// TIA Portal V18 export
// export: Created 2026-01-09T11:32:02.097113Z, ExportSetting WithDefaults, DisplayName Totally Integrated Automation Portal, DisplayVersion V18 Update 5, DisplayName TIA Portal Openness, DisplayVersion V18 Update 5, DisplayName TIA Portal Teamcenter Gateway, DisplayVersion V18, DisplayName TIA Portal Version Control Interface, DisplayVersion V18, DisplayName SINAMICS Startdrive Advanced, DisplayVersion V18 SP2 Update 1, DisplayName SINAMICS Startdrive G110M, G120, G120C, G120D, G120P, G115D, DisplayVersion V18 SP2 Update 1, DisplayName SINAMICS Startdrive G130, G150, S120, S150, SINAMICS MV, S210, G220, S200, DisplayVersion V18 SP2 Update 1, DisplayName STEP 7 Professional, DisplayVersion V18 Update 5, DisplayName STEP 7 Safety, DisplayVersion V18, DisplayName WinCC Professional, DisplayVersion V18 Update 5
TagTable "D"
  DnstDataBlock_DP_Status{0} : Bool  (%DB[SysDDBNum].DBX2.0, CPU S71500-2PN_TP700, 1 s)
  DnstDataBlock_DP_Status{1} : Bool  (%DB[SysDDBNum].DBX2.1, CPU S71500-2PN_TP700, 1 s)
  DnstDataBlock_DP_Status{2} : Bool  (%DB[SysDDBNum].DBX2.2, CPU S71500-2PN_TP700, 1 s)
  DnstDataBlock_DP_Status{3} : Bool  (%DB[SysDDBNum].DBX2.3, CPU S71500-2PN_TP700, 1 s)
  DnstDataBlock_DP_Status{4} : Bool  (%DB[SysDDBNum].DBX2.4, CPU S71500-2PN_TP700, 1 s)
  DnstDataBlock_DP_Status{5} : Bool  (%DB[SysDDBNum].DBX2.5, CPU S71500-2PN_TP700, 1 s)
  DnstDataBlock_DP_Status{6} : Bool  (%DB[SysDDBNum].DBX2.6, CPU S71500-2PN_TP700, 1 s)
  DnstDataBlock_DP_Status{7} : Bool  (%DB[SysDDBNum].DBX2.7, CPU S71500-2PN_TP700, 1 s)
  DnstDataBlock_DP_Status{8} : Bool  (%DB[SysDDBNum].DBX3.0, CPU S71500-2PN_TP700, 1 s)
  DnstDataBlock_DP_Status{9} : Bool  (%DB[SysDDBNum].DBX3.1, CPU S71500-2PN_TP700, 1 s)
  DnstDataBlock_DP_Status{10} : Bool  (%DB[SysDDBNum].DBX3.2, CPU S71500-2PN_TP700, 1 s)
  DnstDataBlock_DP_Status{11} : Bool  (%DB[SysDDBNum].DBX3.3, CPU S71500-2PN_TP700, 1 s)
  DnstDataBlock_DP_Status{12} : Bool  (%DB[SysDDBNum].DBX3.4, CPU S71500-2PN_TP700, 1 s)
  DnstDataBlock_DP_Status{13} : Bool  (%DB[SysDDBNum].DBX3.5, CPU S71500-2PN_TP700, 1 s)
  DnstDataBlock_DP_Status{14} : Bool  (%DB[SysDDBNum].DBX3.6, CPU S71500-2PN_TP700, 1 s)
  DnstDataBlock_DP_Status{15} : Bool  (%DB[SysDDBNum].DBX3.7, CPU S71500-2PN_TP700, 1 s)
  DnstDataBlock_DP_Status{16} : Bool  (%DB[SysDDBNum].DBX4.0, CPU S71500-2PN_TP700, 1 s)
  DnstDataBlock_DP_Status{17} : Bool  (%DB[SysDDBNum].DBX4.1, CPU S71500-2PN_TP700, 1 s)
  DnstDataBlock_DP_Status{18} : Bool  (%DB[SysDDBNum].DBX4.2, CPU S71500-2PN_TP700, 1 s)
  DnstDataBlock_DP_Status{19} : Bool  (%DB[SysDDBNum].DBX4.3, CPU S71500-2PN_TP700, 1 s)
  DnstDataBlock_DP_Status{20} : Bool  (%DB[SysDDBNum].DBX4.4, CPU S71500-2PN_TP700, 1 s)
  DnstDataBlock_DP_Status{21} : Bool  (%DB[SysDDBNum].DBX4.5, CPU S71500-2PN_TP700, 1 s)
  DnstDataBlock_DP_Status{22} : Bool  (%DB[SysDDBNum].DBX4.6, CPU S71500-2PN_TP700, 1 s)
  DnstDataBlock_DP_Status{23} : Bool  (%DB[SysDDBNum].DBX4.7, CPU S71500-2PN_TP700, 1 s)
  DnstDataBlock_DP_Status{24} : Bool  (%DB[SysDDBNum].DBX5.0, CPU S71500-2PN_TP700, 1 s)
  DnstDataBlock_DP_Status{25} : Bool  (%DB[SysDDBNum].DBX5.1, CPU S71500-2PN_TP700, 1 s)
  DnstDataBlock_DP_Status{26} : Bool  (%DB[SysDDBNum].DBX5.2, CPU S71500-2PN_TP700, 1 s)
  DnstDataBlock_DP_Status{27} : Bool  (%DB[SysDDBNum].DBX5.3, CPU S71500-2PN_TP700, 1 s)
  DnstDataBlock_DP_Status{28} : Bool  (%DB[SysDDBNum].DBX5.4, CPU S71500-2PN_TP700, 1 s)
  DnstDataBlock_DP_Status{29} : Bool  (%DB[SysDDBNum].DBX5.5, CPU S71500-2PN_TP700, 1 s)
  DnstDataBlock_DP_Status{30} : Bool  (%DB[SysDDBNum].DBX5.6, CPU S71500-2PN_TP700, 1 s)
  DnstDataBlock_DP_Status{31} : Bool  (%DB[SysDDBNum].DBX5.7, CPU S71500-2PN_TP700, 1 s)
  DnstDataBlock_DP_Status{32} : Bool  (%DB[SysDDBNum].DBX6.0, CPU S71500-2PN_TP700, 1 s)
  DnstDataBlock_DP_Status{33} : Bool  (%DB[SysDDBNum].DBX6.1, CPU S71500-2PN_TP700, 1 s)
  DnstDataBlock_DP_Status{34} : Bool  (%DB[SysDDBNum].DBX6.2, CPU S71500-2PN_TP700, 1 s)
  DnstDataBlock_DP_Status{35} : Bool  (%DB[SysDDBNum].DBX6.3, CPU S71500-2PN_TP700, 1 s)
  DnstDataBlock_DP_Status{36} : Bool  (%DB[SysDDBNum].DBX6.4, CPU S71500-2PN_TP700, 1 s)
  DnstDataBlock_DP_Status{37} : Bool  (%DB[SysDDBNum].DBX6.5, CPU S71500-2PN_TP700, 1 s)
  DnstDataBlock_DP_Status{38} : Bool  (%DB[SysDDBNum].DBX6.6, CPU S71500-2PN_TP700, 1 s)
  DnstDataBlock_DP_Status{39} : Bool  (%DB[SysDDBNum].DBX6.7, CPU S71500-2PN_TP700, 1 s)
  DnstDataBlock_DP_Status{40} : Bool  (%DB[SysDDBNum].DBX7.0, CPU S71500-2PN_TP700, 1 s)
  DnstDataBlock_DP_Status{41} : Bool  (%DB[SysDDBNum].DBX7.1, CPU S71500-2PN_TP700, 1 s)
  DnstDataBlock_DP_Status{42} : Bool  (%DB[SysDDBNum].DBX7.2, CPU S71500-2PN_TP700, 1 s)
  DnstDataBlock_DP_Status{43} : Bool  (%DB[SysDDBNum].DBX7.3, CPU S71500-2PN_TP700, 1 s)
  DnstDataBlock_DP_Status{44} : Bool  (%DB[SysDDBNum].DBX7.4, CPU S71500-2PN_TP700, 1 s)
  DnstDataBlock_DP_Status{45} : Bool  (%DB[SysDDBNum].DBX7.5, CPU S71500-2PN_TP700, 1 s)
  DnstDataBlock_DP_Status{46} : Bool  (%DB[SysDDBNum].DBX7.6, CPU S71500-2PN_TP700, 1 s)
  DnstDataBlock_DP_Status{47} : Bool  (%DB[SysDDBNum].DBX7.7, CPU S71500-2PN_TP700, 1 s)
  DnstDataBlock_DP_Status{48} : Bool  (%DB[SysDDBNum].DBX8.0, CPU S71500-2PN_TP700, 1 s)
  DnstDataBlock_DP_Status{49} : Bool  (%DB[SysDDBNum].DBX8.1, CPU S71500-2PN_TP700, 1 s)
  DnstDataBlock_DP_Status{50} : Bool  (%DB[SysDDBNum].DBX8.2, CPU S71500-2PN_TP700, 1 s)
  DnstDataBlock_DP_Status{51} : Bool  (%DB[SysDDBNum].DBX8.3, CPU S71500-2PN_TP700, 1 s)
  DnstDataBlock_DP_Status{52} : Bool  (%DB[SysDDBNum].DBX8.4, CPU S71500-2PN_TP700, 1 s)
  DnstDataBlock_DP_Status{53} : Bool  (%DB[SysDDBNum].DBX8.5, CPU S71500-2PN_TP700, 1 s)
  DnstDataBlock_DP_Status{54} : Bool  (%DB[SysDDBNum].DBX8.6, CPU S71500-2PN_TP700, 1 s)
  DnstDataBlock_DP_Status{55} : Bool  (%DB[SysDDBNum].DBX8.7, CPU S71500-2PN_TP700, 1 s)
  DnstDataBlock_DP_Status{56} : Bool  (%DB[SysDDBNum].DBX9.0, CPU S71500-2PN_TP700, 1 s)
  DnstDataBlock_DP_Status{57} : Bool  (%DB[SysDDBNum].DBX9.1, CPU S71500-2PN_TP700, 1 s)
  DnstDataBlock_DP_Status{58} : Bool  (%DB[SysDDBNum].DBX9.2, CPU S71500-2PN_TP700, 1 s)
  DnstDataBlock_DP_Status{59} : Bool  (%DB[SysDDBNum].DBX9.3, CPU S71500-2PN_TP700, 1 s)
  DnstDataBlock_DP_Status{60} : Bool  (%DB[SysDDBNum].DBX9.4, CPU S71500-2PN_TP700, 1 s)
  DnstDataBlock_DP_Status{61} : Bool  (%DB[SysDDBNum].DBX9.5, CPU S71500-2PN_TP700, 1 s)
  DnstDataBlock_DP_Status{62} : Bool  (%DB[SysDDBNum].DBX9.6, CPU S71500-2PN_TP700, 1 s)
  DnstDataBlock_DP_Status{63} : Bool  (%DB[SysDDBNum].DBX9.7, CPU S71500-2PN_TP700, 1 s)
  DnstDataBlock_DP_Status{64} : Bool  (%DB[SysDDBNum].DBX10.0, CPU S71500-2PN_TP700, 1 s)
  DnstDataBlock_DP_Status{65} : Bool  (%DB[SysDDBNum].DBX10.1, CPU S71500-2PN_TP700, 1 s)
  DnstDataBlock_DP_Status{66} : Bool  (%DB[SysDDBNum].DBX10.2, CPU S71500-2PN_TP700, 1 s)
  DnstDataBlock_DP_Status{67} : Bool  (%DB[SysDDBNum].DBX10.3, CPU S71500-2PN_TP700, 1 s)
  DnstDataBlock_DP_Status{68} : Bool  (%DB[SysDDBNum].DBX10.4, CPU S71500-2PN_TP700, 1 s)
  DnstDataBlock_DP_Status{69} : Bool  (%DB[SysDDBNum].DBX10.5, CPU S71500-2PN_TP700, 1 s)
  DnstDataBlock_DP_Status{70} : Bool  (%DB[SysDDBNum].DBX10.6, CPU S71500-2PN_TP700, 1 s)
  DnstDataBlock_DP_Status{71} : Bool  (%DB[SysDDBNum].DBX10.7, CPU S71500-2PN_TP700, 1 s)
  DnstDataBlock_DP_Status{72} : Bool  (%DB[SysDDBNum].DBX11.0, CPU S71500-2PN_TP700, 1 s)
  DnstDataBlock_DP_Status{73} : Bool  (%DB[SysDDBNum].DBX11.1, CPU S71500-2PN_TP700, 1 s)
  DnstDataBlock_DP_Status{74} : Bool  (%DB[SysDDBNum].DBX11.2, CPU S71500-2PN_TP700, 1 s)
  DnstDataBlock_DP_Status{75} : Bool  (%DB[SysDDBNum].DBX11.3, CPU S71500-2PN_TP700, 1 s)
  DnstDataBlock_DP_Status{76} : Bool  (%DB[SysDDBNum].DBX11.4, CPU S71500-2PN_TP700, 1 s)
  DnstDataBlock_DP_Status{77} : Bool  (%DB[SysDDBNum].DBX11.5, CPU S71500-2PN_TP700, 1 s)
  DnstDataBlock_DP_Status{78} : Bool  (%DB[SysDDBNum].DBX11.6, CPU S71500-2PN_TP700, 1 s)
  DnstDataBlock_DP_Status{79} : Bool  (%DB[SysDDBNum].DBX11.7, CPU S71500-2PN_TP700, 1 s)
  DnstDataBlock_DP_Status{80} : Bool  (%DB[SysDDBNum].DBX12.0, CPU S71500-2PN_TP700, 1 s)
  DnstDataBlock_DP_Status{81} : Bool  (%DB[SysDDBNum].DBX12.1, CPU S71500-2PN_TP700, 1 s)
  DnstDataBlock_DP_Status{82} : Bool  (%DB[SysDDBNum].DBX12.2, CPU S71500-2PN_TP700, 1 s)
  DnstDataBlock_DP_Status{83} : Bool  (%DB[SysDDBNum].DBX12.3, CPU S71500-2PN_TP700, 1 s)
  DnstDataBlock_DP_Status{84} : Bool  (%DB[SysDDBNum].DBX12.4, CPU S71500-2PN_TP700, 1 s)
  DnstDataBlock_DP_Status{85} : Bool  (%DB[SysDDBNum].DBX12.5, CPU S71500-2PN_TP700, 1 s)
  DnstDataBlock_DP_Status{86} : Bool  (%DB[SysDDBNum].DBX12.6, CPU S71500-2PN_TP700, 1 s)
  DnstDataBlock_DP_Status{87} : Bool  (%DB[SysDDBNum].DBX12.7, CPU S71500-2PN_TP700, 1 s)
  DnstDataBlock_DP_Status{88} : Bool  (%DB[SysDDBNum].DBX13.0, CPU S71500-2PN_TP700, 1 s)
  DnstDataBlock_DP_Status{89} : Bool  (%DB[SysDDBNum].DBX13.1, CPU S71500-2PN_TP700, 1 s)
  DnstDataBlock_DP_Status{90} : Bool  (%DB[SysDDBNum].DBX13.2, CPU S71500-2PN_TP700, 1 s)
  DnstDataBlock_DP_Status{91} : Bool  (%DB[SysDDBNum].DBX13.3, CPU S71500-2PN_TP700, 1 s)
  DnstDataBlock_DP_Status{92} : Bool  (%DB[SysDDBNum].DBX13.4, CPU S71500-2PN_TP700, 1 s)
  DnstDataBlock_DP_Status{93} : Bool  (%DB[SysDDBNum].DBX13.5, CPU S71500-2PN_TP700, 1 s)
  DnstDataBlock_DP_Status{94} : Bool  (%DB[SysDDBNum].DBX13.6, CPU S71500-2PN_TP700, 1 s)
  DnstDataBlock_DP_Status{95} : Bool  (%DB[SysDDBNum].DBX13.7, CPU S71500-2PN_TP700, 1 s)
  DnstDataBlock_DP_Status{96} : Bool  (%DB[SysDDBNum].DBX14.0, CPU S71500-2PN_TP700, 1 s)
  DnstDataBlock_DP_Status{97} : Bool  (%DB[SysDDBNum].DBX14.1, CPU S71500-2PN_TP700, 1 s)
  DnstDataBlock_DP_Status{98} : Bool  (%DB[SysDDBNum].DBX14.2, CPU S71500-2PN_TP700, 1 s)
  DnstDataBlock_DP_Status{99} : Bool  (%DB[SysDDBNum].DBX14.3, CPU S71500-2PN_TP700, 1 s)
  DnstDataBlock_DP_Status{100} : Bool  (%DB[SysDDBNum].DBX14.4, CPU S71500-2PN_TP700, 1 s)
  DnstDataBlock_DP_Status{101} : Bool  (%DB[SysDDBNum].DBX14.5, CPU S71500-2PN_TP700, 1 s)
  DnstDataBlock.DP.Index : Word  (%DB[SysDDBNum].DBW0, CPU S71500-2PN_TP700, 1 s)
